/// Enable/Disable robot into RA power state "Enabled"
FUNCTION_BLOCK EnableRobotFB EXTENDS RobotLibraryBaseFB
// ------------------------------------------------------------------------- 
//  SRCI Robot Library                                                
// ------------------------------------------------------------------------- 
//                                                                           
//  Object:      EnableRobotFB                                       
//  Author:      Thorsten Brach                                                
//  Date:        2024-06-01
//
//  Description:                                              
//   
//                                                                           
//  Copyright: 
//    (C) 2024 Thorsten Brach. All rights reserved                                                                         
//                                                                           
//  Disclaimer:                                                                           
//    This project is provided without any guarantee and can be used for   
//    private and commercial purposes. Any commercial use is at the user’s 
//    own risk and responsibility.
//
// -------------------------------------------------------------------------
VAR_INPUT
  /// Set TRUE to change RA power state to "Enabled"
  Enable            : BOOL;
  /// Command parameter 
  ParCmd            : EnableRobotParCmd;
END_VAR


VAR_OUTPUT
  /// command results
  OutCmd            : EnableRobotOutCmd;
  /// FB is being processed
  Busy              : BOOL;
  /// Command is transferred and confirmed by the RC
  CommandBuffered   : BOOL;
  /// Receiving of input parameter values has been acknowledged by RC
  ParameterAccepted : BOOL;
END_VAR

VAR
  /// internal copy of command parameter 
 _parCmd            : EnableRobotParCmd;
  /// command data to send
 _command           : EnableRobotSendData;
  /// response data received
 _response          : EnableRobotRecvData;
  /// Rising edge for enable
 _enable_R          : R_TRIG;
  /// Falling edge for enable
 _enable_F          : R_TRIG;

END_VAR

                  

                

METHOD CheckParameterChanged : BOOL
                        // compare memory 
CheckParameterChanged := ( MemCmp(ADR(ParCmd), ADR(_parCmd), SIZEOF(ParCmd)) = RobotLibraryConstants.OK );

IF ( CheckParameterChanged )
THEN  
  // update internal copy of parameters 
 _parCmd := ParCmd;
  // inc parameter sequence
 _command.ParSeq := _command.ParSeq + 1;
  // update command data  
  CommandData := CreateCommandData(); // ( Access via reference to rCommandFB in ACR )
END_IF
                      
END_METHOD

METHOD CreateCommandData : SendData
                        // Table 6-25: Sent CMD payload (PLC to RC) of "EnableRobot"

// --------------------------
// Header
// --------------------------
// Byte 00 : UINT  - Type HB     
// Byte 01 :       - Type LB    
// Byte 02 : USINT - Reserve | ExecutionMode
// Byte 03 : USINT - ParSeq  | Priority
// --------------------------
// Datablock
// --------------------------
// Byte 04 : BOOL  - Enable
// Byte 05 : BOOL  - HoldToRun
// Byte 06 : USINT - StepMode   
// Byte 07 : BOOL  - ManualStep
// --------------------------

// set command parameter 
_command.CmdTyp    :=  CmdType.EnableRobot;
_command.ExecMode  :=  ExecutionMode.PARALLEL;
_command.ParSeq    := _command.ParSeq;
_command.Priority  :=  PriorityLevel.NORMAL;
_command.Enable    :=  Enable;
_command.HoldToRun := _parCmd.HoldToRun;
_command.StepMode  := _parCmd.StepMode;
_command.ManualStep:= _parCmd.ManualStep;


// copy command data to header
_cmdHeader := _command;
// call base implementation to copy header to payload buffer
SUPER^.CreateCommandData();

// add command.Enable
CreateCommandData.AddBool(_command.Enable);
// add command.StepMode
CreateCommandData.AddByte(_command.StepMode);
// add command.HoldToRun
CreateCommandData.AddBool(_command.HoldToRun);
// add command.ManualStep
CreateCommandData.AddBool(_command.ManualStep);
                      
END_METHOD

METHOD PROTECTED OnCall
VAR_IN_OUT
  /// Robot assignment of function
  AxesGroup : AxesGroup; 
END_VAR
                        // building rising and falling edges
_enable_R( CLK := Enable);
_enable_F( CLK := Enable);

CASE _stepCmd OF
  
  00:  IF ( _enable_R.Q ) OR (_enable_F.Q) 
       THEN
         // set busy flag
         Busy := TRUE;
         // Reset command outputs
         MemSet(ADR(OutCmd),0,SIZEOF(OutCmd));         
         // apply command parameter
        _parCmd := ParCmd;
         // init parameter sequence
        _command.ParSeq := 1;
         // set timeout
         SetTimeout(PT := _timeoutCmd, rTimer := _timerCmd);
         // inc step counter
        _stepCmd := _stepCmd + 1; 
	     END_IF
     
  01:  // create command data
       CommandData := CreateCommandData();
       // Add command to active command register
      _uniqueID := AxesGroup.Acyclic.ActiveCommandRegister.AddCmd( rCommandFB := THIS^ );     
       // set timeout
       SetTimeout(PT := _timeoutCmd, rTimer := _timerCmd);
       // inc step counter
      _stepCmd := _stepCmd + 1; 

  02:  // Wait for responce received
       IF ( _responseReceived )
       THEN
         // reset response received flag
        _responseReceived := FALSE;

         CASE  _response.State 
         OF
           CmdMessageState.BUFFERED    : CommandBuffered    := TRUE;
           CmdMessageState.ERROR       : Error              := TRUE;
				 END_CASE
                
         // Done, Aborted or Error ?
         IF (_response.State >= CmdMessageState.DONE )
         THEN
           // Update results
           OutCmd.Enabled     := _response.Enabled;
           // set timeout
           SetTimeout(PT := _timeoutCmd, rTimer := _timerCmd);
           // inc step counter
          _stepCmd := _stepCmd + 1; 
				 END_IF
       END_IF

  03: // reset step counter
     _stepCmd := 0;
      // reset busy flag
      Busy := FALSE;    
      // reset buffered flag
      CommandBuffered := FALSE;  
ELSE
  // invalid step
  ErrorID := RobotLibraryEvents.ERR_INVALID_STEP;
END_CASE



// Reset FB
IF ( FALSE ) {warning 'ToDo: find condition'}
THEN
 _uniqueId           := 0;
 _stepCmd            := 0;
  Busy               := FALSE;
  CommandBuffered    := FALSE;
  Error              := FALSE;
  ErrorID            := 0;
  WarningID          := 0;
  InfoID             := 0;  
END_IF
                      
END_METHOD

METHOD ParseResponsePayload : DINT
VAR_INPUT
  /// Response data
  ResponseData : RecvData;
END_VAR
VAR
 /// index for payload buffer
 _idx : DINT;  
END_VAR
                        // Table 6-26: Received CMD payload (RC to PLC) of "EnableRobot"
// --------------------------
// Header
// --------------------------
// Byte 00 : USINT - ParSeq | State     
// Byte 01 : SINT  - AlarmMessageSeverity    
// Byte 02 : UINT  - AlarmMessageCode HB
// Byte 03 :       - AlarmMessageCode LB
// --------------------------
// Datablock
// --------------------------
// Byte 04 : BOOL  - Enabled
// --------------------------

// call base implementation to parse the header from payload buffer
SUPER^.ParseResponseData(ResponseData);

// copy parsed header to response
_response.ParSeq               := _rspHeader.ParSeq;
_response.State                := _rspHeader.State;
_response.AlarmMessageSeverity := _rspHeader.AlarmMessageSeverity;
_response.AlarmMessageCode     := _rspHeader.AlarmMessageCode;

// Get Response.Enabled
_response.Enabled := ResponseData.GetBool();
                      
END_METHOD
END_FUNCTION_BLOCK

/// Calculate Forward Kinematic
FUNCTION_BLOCK CalculateForwardKinematicFB EXTENDS RobotLibraryBaseFB
// ------------------------------------------------------------------------- 
//  SRCI Robot Library                                                
// ------------------------------------------------------------------------- 
//                                                                           
//  Object:      CalculateForwardKinematicFB                                       
//  Author:      Thorsten Brach                                                
//  Date:        2024-06-01
//
//  Description:                                              
//   
//                                                                           
//  Copyright: 
//    (C) 2024 Thorsten Brach. All rights reserved                                                                         
//                                                                           
//  Disclaimer:                                                                           
//    This project is provided without any guarantee and can be used for   
//    private and commercial purposes. Any commercial use is at the user’s 
//    own risk and responsibility.
//
// -------------------------------------------------------------------------
VAR_INPUT
  /// Start of the command at the rising edge
  Execute            : BOOL;
  /// Command parameter 
  ParCmd             : CalculateForwardKinematicParCmd;    
END_VAR
VAR_OUTPUT
  /// The command has been completed successfully
  Done               : BOOL;
  /// FB is being processed
  Busy               : BOOL;
  /// Command is transferred and confirmed by the RC
  CommandBuffered    : BOOL;
  /// Command output 
  OutCmd            : CalculateForwardKinematicOutCmd;  
END_VAR

VAR
  /// internal copy of command parameter 
 _parCmd             : CalculateForwardKinematicParCmd;
  /// command data to send
 _command            : CalculateForwardKinematicSendData;
  /// response data received
 _response           : CalculateForwardKinematicRecvData;      
END_VAR

                  
                

METHOD CheckParameterChanged : BOOL
                        // compare memory 
CheckParameterChanged := ( MemCmp(ADR(ParCmd), ADR(_parCmd), SIZEOF(ParCmd)) = RobotLibraryConstants.OK );

IF ( CheckParameterChanged )
THEN  
  // update internal copy of parameters 
 _parCmd := ParCmd;
  // inc parameter sequence
 _command.ParSeq := _command.ParSeq + 1;
  // update command data  
  CommandData := CreateCommandData(); // ( Access via reference to rCommandFB in ACR )
END_IF
                      
END_METHOD

METHOD CreateCommandData : SendData
                        // Table 6-681: Sent CMD payload (PLC to RC) of "OpenBrake"

// --------------------------
// Header
// --------------------------
// Byte 00 : UINT  - Type HB     
// Byte 01 :       - Type LB    
// Byte 02 : USINT - Reserve | ExecutionMode
// Byte 03 : USINT - ParSeq  | Priority
// --------------------------
// Datablock
// --------------------------
// Byte 04 : BYTE - RobotAxesBrakeRelease
// Byte 05 : BYTE - ExternalAxesBrakeRelease
// --------------------------

// set command parameter 
_command.CmdTyp                     :=  CmdType.CalculateForwardKinematic;
_command.ExecMode                   :=  ExecutionMode.PARALLEL;
_command.ParSeq                     := _command.ParSeq;
_command.Priority                   :=  PriorityLevel.NORMAL;
_command.ToolNo                     := _parCmd.ToolNo;
_command.FrameNo                    := _parCmd.FrameNo;
_command.CartesianPosition          := _parCmd.CartesianPosition;

// copy command data to header
_cmdHeader := _command;
// call base implementation to copy header to payload buffer
SUPER^.CreateCommandData();

// add command.ToolNo
CreateCommandData.AddUsint(_command.ToolNo);
// add command.FrameNo
CreateCommandData.AddUsint(_command.FrameNo);
// add command.CartesianPosition.X
CreateCommandData.AddReal(_command.CartesianPosition.X);
// add command.CartesianPosition.Y
CreateCommandData.AddReal(_command.CartesianPosition.Y);
// add command.CartesianPosition.Z
CreateCommandData.AddReal(_command.CartesianPosition.Z);
// add command.CartesianPosition.Rx
CreateCommandData.AddReal(_command.CartesianPosition.Rx);
// add command.CartesianPosition.Ry
CreateCommandData.AddReal(_command.CartesianPosition.Ry);
// add command.CartesianPosition.Rz
CreateCommandData.AddReal(_command.CartesianPosition.Rz);
// add command.CartesianPosition.E1
CreateCommandData.AddReal(_command.CartesianPosition.E1);
// add command.CartesianPosition.E2
CreateCommandData.AddReal(_command.CartesianPosition.E2);
// add command.CartesianPosition.E3
CreateCommandData.AddReal(_command.CartesianPosition.E3);
// add command.CartesianPosition.E4
CreateCommandData.AddReal(_command.CartesianPosition.E4);
// add command.CartesianPosition.E5
CreateCommandData.AddReal(_command.CartesianPosition.E5);
// add command.CartesianPosition.E6
CreateCommandData.AddReal(_command.CartesianPosition.E6);
                      
END_METHOD

METHOD PROTECTED OnCall
VAR_IN_OUT
  /// Robot assignment of function
  AxesGroup : AxesGroup; 
END_VAR
                        CASE _stepCmd OF
  
  00:  IF ( Execute ) 
       THEN
         // set busy flag
         Busy := TRUE;
         // Reset command outputs
         MemSet(ADR(OutCmd),0,SIZEOF(OutCmd));         
         // apply command parameter
        _parCmd := ParCmd;
         // init parameter sequence
        _command.ParSeq := 1;
         // set timeout
         SetTimeout(PT := _timeoutCmd, rTimer := _timerCmd);
         // inc step counter
        _stepCmd := _stepCmd + 1; 
	     END_IF
     
  01:  // create command data
       CommandData := CreateCommandData();
       // Add command to active command register
      _uniqueID := AxesGroup.Acyclic.ActiveCommandRegister.AddCmd( rCommandFB := THIS^ );     
       // set timeout
       SetTimeout(PT := _timeoutCmd, rTimer := _timerCmd);
       // inc step counter
      _stepCmd := _stepCmd + 1; 

  02:  // Wait for responce received
       IF ( _responseReceived )
       THEN
         // reset response received flag
        _responseReceived := FALSE;

         CASE  _response.State 
         OF
           CmdMessageState.BUFFERED    : CommandBuffered    := TRUE;
           CmdMessageState.ERROR       : Error              := TRUE;
				 END_CASE
                
         // Done, Aborted or Error ?
         IF (_response.State >= CmdMessageState.DONE )
         THEN
           // Update results
           OutCmd.TargetToolNoReturn      := _response.TargetToolNoReturn;
           OutCmd.TargetFrameNoReturn     := _response.TargetFrameNoReturn;
           OutCmd.CartesianPosition       := _response.CartesianPosition;

           // set timeout
           SetTimeout(PT := _timeoutCmd, rTimer := _timerCmd);
           // inc step counter
          _stepCmd := _stepCmd + 1; 
				 END_IF
       END_IF

  03: Done := TRUE;
      IF ( NOT Execute)
      THEN
        // reset step counter
       _stepCmd := 0;
        // reset done flag
        Done := FALSE;
        // reset busy flag
        Busy := FALSE; 
        // reset buffered flag
        CommandBuffered := FALSE;  
			END_IF     
ELSE
  // invalid step
  ErrorID := RobotLibraryEvents.ERR_INVALID_STEP;
END_CASE


// Cancel 
IF (Busy) AND (NOT Execute) 
THEN
  // try to remove cmd
  AxesGroup.Acyclic.ActiveCommandRegister.RemoveCmd(_uniqueID);
END_IF


// Reset FB
IF ( NOT Execute )
THEN
 _uniqueId           := 0;
 _stepCmd            := 0;
  Done               := FALSE;
  Busy               := FALSE;
  CommandBuffered    := FALSE;
  Error              := FALSE;
  ErrorID            := 0;
  WarningID          := 0;
  InfoID             := 0;  
END_IF
                      
END_METHOD

METHOD ParseResponsePayload : DINT
VAR_INPUT
  /// Response data
  ResponseData : RecvData;
END_VAR
                        // Table 6-741: Received CMD payload (RC to PLC) of "BrakeTest"
// --------------------------
// Header
// --------------------------
// Byte 00 : USINT - ParSeq | State     
// Byte 01 : SINT  - AlarmMessageSeverity    
// Byte 02 : UINT  - AlarmMessageCode HB
// Byte 03 :       - AlarmMessageCode LB
// --------------------------
// Datablock
// --------------------------
// Byte 04 : BOOL  - Enabled
// Byte 05 : BYTE  - RobotAxesBrakeReleased
// Byte 06 : BYTE  - ExternalAxesBrakeReleased
// --------------------------

// call base implementation to parse the header from payload buffer
SUPER^.ParseResponseData(ResponseData);

// copy parsed header to response
_response.ParSeq               := _rspHeader.ParSeq;
_response.State                := _rspHeader.State;
_response.AlarmMessageSeverity := _rspHeader.AlarmMessageSeverity;
_response.AlarmMessageCode     := _rspHeader.AlarmMessageCode;

// Get TargetToolNoReturn
_response.TargetToolNoReturn   := ResponseData.GetUsint();
// Get TargetFrameNoReturn
_response.TargetFrameNoReturn  := ResponseData.GetUsint();
// Get CartesianPosition.X
_response.CartesianPosition.X := ResponseData.GetReal();
// Get CartesianPosition.Y
_response.CartesianPosition.Y := ResponseData.GetReal();
// Get CartesianPosition.Z
_response.CartesianPosition.Z := ResponseData.GetReal();
// Get CartesianPosition.Rx
_response.CartesianPosition.Rx := ResponseData.GetReal();
// Get CartesianPosition.Ry
_response.CartesianPosition.Ry := ResponseData.GetReal();
// Get CartesianPosition.Rz
_response.CartesianPosition.Rz := ResponseData.GetReal();
// Get CartesianPosition.Config
_response.CartesianPosition.Config := ResponseData.GetArmConfig();
// Get CartesianPosition.TurnNumber
_response.CartesianPosition.TurnNumber := ResponseData.GetTurnNumbers();
// Get CartesianPosition.E1
_response.CartesianPosition.E1 := ResponseData.GetReal();
// Get CartesianPosition.E2
_response.CartesianPosition.E2 := ResponseData.GetReal();
// Get CartesianPosition.E3
_response.CartesianPosition.E3 := ResponseData.GetReal();
// Get CartesianPosition.E4
_response.CartesianPosition.E4 := ResponseData.GetReal();
// Get CartesianPosition.E5
_response.CartesianPosition.E5 := ResponseData.GetReal();
// Get CartesianPosition.E6
_response.CartesianPosition.E6 := ResponseData.GetReal();

                      
END_METHOD
END_FUNCTION_BLOCK

CONFIGURATION Application
  RESOURCE RobotLibrary ON PLC
(* global variable list RobotLibraryEvents *)
{attribute 'qualified_only'}
VAR_GLOBAL
  /// Program fault : Invalid step
  ERR_INVALID_STEP : WORD := 1;
END_VAR
(* global variable list RobotLibraryConstants *)
{attribute 'qualified_only'}
// ------------------------------------------------------------------------- 
//  SRCI Robot Library                                                
// ------------------------------------------------------------------------- 
//                                                                           
//  Object:      RobotLibraryConstants                                       
//  Author:      Thorsten Brach                                                
//  Date:        2024-06-01
//
//  Description:                                              
//   
//                                                                           
//  Copyright: 
//    (C) 2024 Thorsten Brach. All rights reserved                                                                         
//                                                                           
//  Disclaimer:                                                                           
//    This project is provided without any guarantee and can be used for   
//    private and commercial purposes. Any commercial use is at the user’s 
//    own risk and responsibility.
//
// -------------------------------------------------------------------------
VAR_GLOBAL CONSTANT
  /// Minimal amount of tools
  TOOL_MIN             : DINT :=  16;
  /// Maximal amount of tools
  TOOL_MAX             : DINT := 255;
  /// Minimal amount of frames
  FRAME_MIN            : DINT :=  16;
  /// Maximal amount of frames
  FRAME_MAX            : DINT := 255;
  /// Minimal amount of loads
  LOAD_MIN             : DINT :=  16;  
  /// Maximal amount of loads
  LOAD_MAX             : DINT := 255;  
  /// Minimal amount of work areas
  WORK_AREAS_MIN       : DINT :=   8;  
  /// Maximal amount of work areas
  WORK_AREAS_MAX       : DINT := 255;  
  /// Maximal amount of bytes which are allowed to be exchanged with the sub program of the RC
  SUB_PROGRAM_DATA_MAX : DINT := 190;

  /// Version of SRCI specification
  /// Bit 0-4 : Minor version = Features        (0..31)
  /// Bit 5-7 : Major version = Breaking change (0..07)
  SRCIVersion            : VersionStruct := ( MajorVersion := 0, MinorVersion := 1, PatchVersion := 0);

  /// OK = 0
  OK                   : DINT := 0;
  /// Running = 1
  RUNNING              : DINT := 1;
END_VAR
(* global variable list RobotLibraryParameter *)
{attribute 'qualified_only'}
// ------------------------------------------------------------------------- 
//  SRCI Robot Library                                                
// ------------------------------------------------------------------------- 
//                                                                           
//  Object:      Parameter                                       
//  Author:      Thorsten Brach                                                
//  Date:        2024-06-01
//
//  Description:                                              
//   
//                                                                           
//  Copyright: 
//    (C) 2024 Thorsten Brach. All rights reserved                                                                         
//                                                                           
//  Disclaimer:                                                                           
//    This project is provided without any guarantee and can be used for   
//    private and commercial purposes. Any commercial use is at the user’s 
//    own risk and responsibility.
//
// -------------------------------------------------------------------------
VAR_GLOBAL CONSTANT
  /// Maximal amount of input data
  ROBOT_IN_DATA_MAX                   : UINT := 255;
  /// Maximal amount of output data
  ROBOT_OUT_DATA_MAX                  : UINT := 255;
  /// Maximal amount of tools
  TOOL_MAX                            : DINT := 255;
  /// Maximal amount of frames
  FRAME_MAX                           : DINT := 255;
  /// Maximal amount of loads
  LOAD_MAX                            : DINT := 255;  
  /// Maximal amount of work areas
  WORK_AREAS_MAX                      : DINT := 255;  
  /// Maximal amount of system logs
  SYSTEM_LOG_MAX                      : DINT := 32;  
  /// Maximal amount of message logs
  MESSAGE_LOG_MAX                     : DINT := 32;  
  /// Maximal amount of List entries 
  LIST_ENTRIES_MAX                    : DINT := 100;
  /// Maximal amount of bytes for the telegram payload
  TELEGRAM_PAYLOAD_MAX                : DINT := 255;  
  /// Maximal amount of bytes for the parameter payload
  PARAMETER_PAYLOAD_MAX               : DINT := 128;  
  /// Maximal amount of bytes for the response payload
  RESPONSE_PAYLOAD_MAX                : DINT := 128;  
  /// Maximal amount of bytes that can be exchanged with the sub program on the RC
  SUB_PROGRAM_DATA_MAX                : DINT := 64;
  /// Maximal amount of spline data
  SPLINE_DATA_MAX                     : DINT := 64;
  /// Maximal amount of entries in the Active Command Register
  ACTIVE_CMD_REGISTER_ENTRIES_MAX     : DINT := 50;
  
  /// Flag to indicate that the byte order must be changed
  SWAP_BYTE_ORDER                     : BOOL := TRUE; {warning 'ToDo: Detect local byte order'}

END_VAR
  END_RESOURCE
END_CONFIGURATION
